TYPE T_DB_LongSTRING : STRING(1024);
END_TYPE

(* stored: Version 1.1.0.1
   DUT T_DB_LongSTRING: Id {28dd9b0e-334a-4690-92a8-f42cd8f9b55d} *)
